// TIA Portal V17 export
// export: Created 2023-12-22T15:03:18.7490077Z, ExportSetting WithDefaults, DisplayName Totally Integrated Automation Portal, DisplayVersion V17, DisplayName TIA Portal Openness, DisplayVersion V17, DisplayName TIA Portal Version Control Interface, DisplayVersion V17, DisplayName STEP 7 Professional, DisplayVersion V17, DisplayName STEP 7 Safety, DisplayVersion V17, DisplayName WinCC Advanced, DisplayVersion V17
DATA_BLOCK "Main_Logick_DB"   // DB1
VERSION : 0.1
// stored: AutoNumber true, DBAccessibleFromOPCUA true, DBAccessibleFromWebserver true, InstanceOfName Main_Logick, InstanceOfType FB
"Main_Logick"
   // VAR RETAIN
   //    Time_Contrast_SKV { S7_SetPoint := 'True'} : "Time_D";
   // END_VAR
BEGIN
   Time_Contrast_SKV.SP_D := 3;
   Time_Contrast_SKV.SP_H := 0;
   Time_Contrast_SKV.SP_M := 0;
   Time_Contrast_SKV.SP_S := 0;
END_DATA_BLOCK
